SUBAPPLICATION Uebung_010d2_sub_AX (* Toggle Flip-Flop mit IE SoftKey_F1 SK_RELEASED mit GreenWhiteBackground *)
  (* Standard: 61499-2; Description: Copyright (c) 2026 Meisterschulen am Ostbahnhof This program and the accompanying materials are made available under the terms of the Eclipse Public License 2.0 which is available at https://www.eclipse.org/legal/epl-2.0/ SPDX-License-Identifier: EPL-2.0 *)
  (* Version 1.0, 2026-09-02, Franz Höpfinger, Meisterschulen am Ostbahnhof, initial API and implementation and/or initial documentation *)
  PACKAGE Uebungen;
  IMPORT Uebungen::const::UT::DefaultPool::SoftKey_F1;
  IMPORT logiBUS::io::DQ::logiBUS_DO;
  IMPORT logiBUS::io::DQ::logiBUS_DO_S;
  IMPORT isobus::UT::io::Softkey::SoftKeyActivationCode::SK_RELEASED;
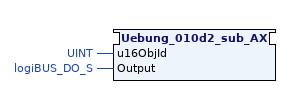
  VAR_INPUT
    u16ObjId : UINT := SoftKey_F1; (* Object ID *)
    Output : logiBUS::io::DQ::logiBUS_DO_S := logiBUS_DO::Output_Q1; (* Identify the Output Output_Q1..Q8 *)
  END_VAR
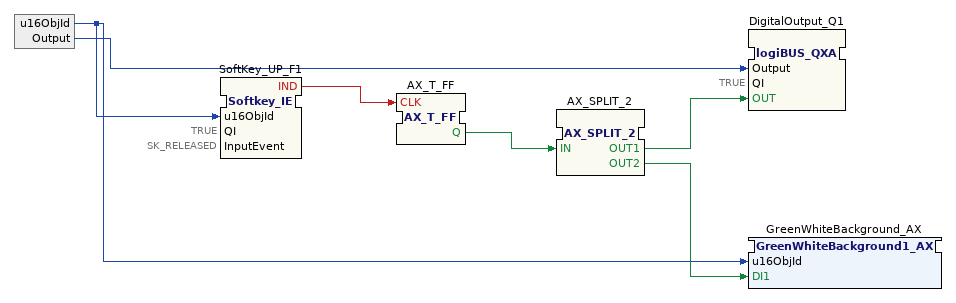
  FBS
    SoftKey_UP_F1 : isobus::UT::io::Softkey::Softkey_IE(QI := TRUE, InputEvent := SK_RELEASED);
    AX_T_FF : adapter::events::unidirectional::AX_T_FF;
    AX_SPLIT_2 : adapter::events::unidirectional::AX_SPLIT_2;
    DigitalOutput_Q1 : logiBUS::io::DQ::logiBUS_QXA(QI := TRUE);
  END_FBS
  SUBAPPS
    GreenWhiteBackground_AX : MyLib::sys::GreenWhiteBackground1_AX;
  END_SUBAPPS
  EVENT_CONNECTIONS
    SoftKey_UP_F1.IND TO AX_T_FF.CLK;
  END_CONNECTIONS
  DATA_CONNECTIONS
    u16ObjId TO SoftKey_UP_F1.u16ObjId;
    u16ObjId TO GreenWhiteBackground_AX.u16ObjId;
    Output TO DigitalOutput_Q1.Output;
  END_CONNECTIONS
  ADAPTER_CONNECTIONS
    AX_T_FF.Q TO AX_SPLIT_2.IN;
    AX_SPLIT_2.OUT1 TO DigitalOutput_Q1.OUT;
    AX_SPLIT_2.OUT2 TO GreenWhiteBackground_AX.DI1;
  END_CONNECTIONS
END_SUBAPPLICATION
